// TIA Portal project "SortingLine_Project" (V18)

(* hardware
DEVICE "S7-1200 station_1"  S7-1200 Station
   slot 0: "Rack_0"  S7-1200 Rack  Rack  V1.0
   slot 1: "PLC_Sorting"  CPU 1214C DC/DC/DC  6ES7 214-1AG40-0XB0  V4.6
*)

// ===== PLC "PLC_Sorting"  CPU 1214C DC/DC/DC =====

VAR_GLOBAL   // PLC tag table "Default tag table"
   "start_button" AT %I100.0 : Bool;   // Start push button, NO
   "stop_button" AT %I100.1 : Bool;   // Stop push button, NC
   "emergency_stop" AT %I100.2 : Bool;   // Emergency stop, NC
   "mode_auto" AT %I100.3 : Bool;   // Mode selector, 1 for auto, 0 for manual
   "sensor_entry" AT %I100.4 : Bool;   // Entry sensor, box presence detection
   "sensor_size_low" AT %I100.5 : Bool;   // Low size sensor, detects small boxes
   "sensor_size_high" AT %I100.6 : Bool;   // High size sensor, detects large boxes
   "sensor_left_entry" AT %I100.7 : Bool;   // Pusher 1 retracted limit switch
   "sensor_evac_lane_1" AT %I101.0 : Bool;   // Lane 1 evacuation sensor
   "sensor_evac_lane_2" AT %I101.1 : Bool;   // Lane 2 evacuation sensor
   "light_green" AT %Q0.0 : Bool;   // Green light, machine running
   "light_red" AT %Q0.1 : Bool;   // Red light, machine stopped or fault
   "motor_main_conveyor" AT %Q0.2 : Bool;   // Main conveyor motor
   "motor_lane_1" AT %Q0.3 : Bool;   // Lane 1 conveyor motor
   "motor_lane_2" AT %Q0.4 : Bool;   // Lane 2 conveyor motor
   "pusher_1_command" AT %Q0.5 : Bool;   // Pusher 1 command
   "pusher_2_command" AT %Q0.6 : Bool;   // Pusher 2 command
   "system_running" AT %M0.0 : Bool;   // System running state
   "system_fault" AT %M0.1 : Bool;   // System in fault state
   "box_detected" AT %M0.2 : Bool;   // A box is currently detected
   "box_is_small" AT %M0.3 : Bool;   // Current box is small
   "box_is_large" AT %M0.4 : Bool;   // Current box is large
   "start_pulse" AT %M1.0 : Bool;   // One scan pulse on rising edge of Start_Button
   "edge_start" AT %M1.1 : Bool;   // Edge memory bit for the P_TRIG instruction
   "edge_entry" AT %M1.2 : Bool;
   "edge_evac_lane_1" AT %M1.3 : Bool;
   "edge_evac_lane_2" AT %M1.4 : Bool;
   "entry_pulse" AT %M1.5 : Bool;
   "evac_lane_1_pulse" AT %M1.6 : Bool;
   "evac_lane_2_pulse" AT %M1.7 : Bool;
   "alignment_done" AT %M2.0 : Bool;
   "counter_lane_1" AT %MW10 : Int;
   "counter_lane_2" AT %MW12 : Int;
   "reset_button" AT %I101.2 : Bool;
   "sensor_load_position" AT %I101.3 : Bool;
   "sensor_unload_position" AT %I101.4 : Bool;
   "reset_light" AT %Q0.7 : Bool;
   "motor_feeder" AT %Q1.0 : Bool;
   "light_yellow" AT %Q1.1 : Bool;
   "turn_command" AT %Q1.2 : Bool;
END_VAR

DATA_BLOCK "FB_Mode_Manager_DB"   // DB1
{ S7_Optimized_Access := 'TRUE' }
VERSION : 0.1
// stored: InstanceOfName FB_Mode_Manager
"FB_Mode_Manager"
BEGIN
END_DATA_BLOCK

DATA_BLOCK "FB_Sorting_Logic_DB"   // DB2
{ S7_Optimized_Access := 'TRUE' }
VERSION : 0.1
// stored: InstanceOfName FB_Sorting_Logic
"FB_Sorting_Logic"
BEGIN
END_DATA_BLOCK

DATA_BLOCK "DB_Global"   // DB3
{ S7_Optimized_Access := 'TRUE' }
VERSION : 0.1
BEGIN
END_DATA_BLOCK

// folder: System blocks/Program resources

DATA_BLOCK "Timer_Alignment"   // DB4
{ S7_Optimized_Access := 'TRUE' }
AUTHOR : Simatic
FAMILY : IEC
NAME : IEC_TMR
VERSION : 1.0
// stored: InstanceOfName IEC_TIMER
"IEC_TIMER"
BEGIN
END_DATA_BLOCK

// folder: (top level)

FUNCTION_BLOCK "FB_Mode_Manager"   // FB1, LAD
{ S7_Optimized_Access := 'TRUE' }
VERSION : 0.1
// FB_Mode_Manager
// Purpose: manage safety, mode selection, start and stop logic, indicator lights, main conveyor motor command.
// Inputs: Start_Button, Stop_Button, Emergency_Stop, Mode_Auto
// Outputs: System_Running, System_Fault, Motor_Main_Conveyor, Light_Green, Light_Red
// Author: HoraEmbedded
// Date: 29/09/26
   VAR_TEMP   // added for the SCL form of the ladder/FBD networks
      _w1 : Bool;
   END_VAR
BEGIN

REGION Network 1: Rising edge detection on Start
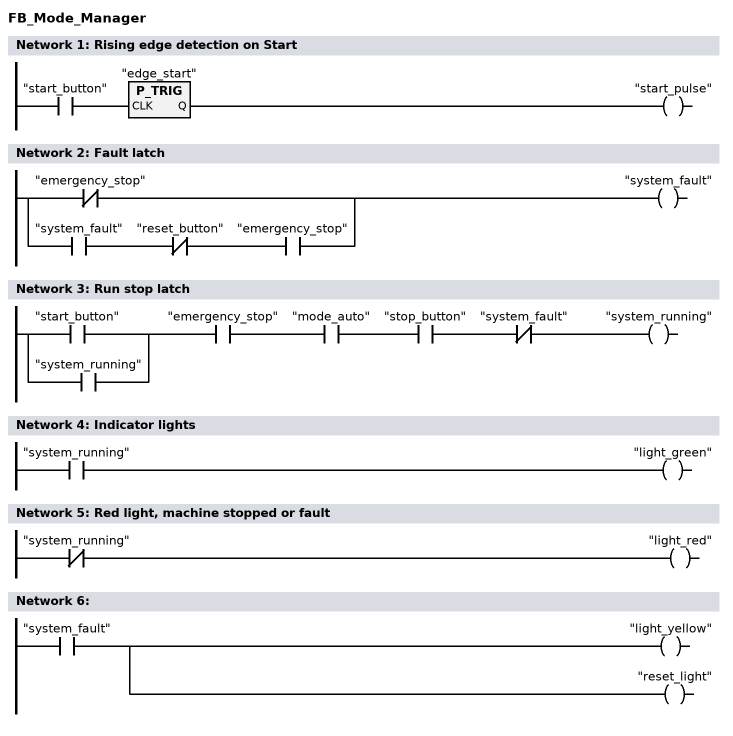
   RUNG wire#powerrail
      Contact( "start_button" )
      P_Trig( "edge_start" )
      Coil( "start_pulse" )
   END_RUNG
   // the same network as SCL:
   #_w1 := "start_button" AND NOT "edge_start";   // rising edge
   "edge_start" := "start_button";
   "start_pulse" := #_w1;
END_REGION

REGION Network 2: Fault latch
   RUNG wire#powerrail
      I_Contact( "emergency_stop" )
      wire#w1
      Coil( "system_fault" )
   END_RUNG
   RUNG wire#powerrail
      Contact( "system_fault" )
      I_Contact( "reset_button" )
      Contact( "emergency_stop" )
   END_RUNG wire#w1
   // the same network as SCL:
   "system_fault" := NOT "emergency_stop" OR ("system_fault" AND NOT "reset_button" AND "emergency_stop");
END_REGION

REGION Network 3: Run stop latch
   RUNG wire#powerrail
      Contact( "start_button" )
      wire#w1
      Contact( "emergency_stop" )
      Contact( "mode_auto" )
      Contact( "stop_button" )
      I_Contact( "system_fault" )
      Coil( "system_running" )
   END_RUNG
   RUNG wire#powerrail
      Contact( "system_running" )
   END_RUNG wire#w1
   // the same network as SCL:
   "system_running" := ("start_button" OR "system_running") AND "emergency_stop" AND "mode_auto" AND "stop_button" AND NOT "system_fault";
END_REGION

REGION Network 4: Indicator lights
   RUNG wire#powerrail
      Contact( "system_running" )
      Coil( "light_green" )
   END_RUNG
   // the same network as SCL:
   "light_green" := "system_running";
END_REGION

REGION Network 5: Red light, machine stopped or fault
   RUNG wire#powerrail
      I_Contact( "system_running" )
      Coil( "light_red" )
   END_RUNG
   // the same network as SCL:
   "light_red" := NOT "system_running";
END_REGION

REGION Network 6
   RUNG wire#powerrail
      Contact( "system_fault" )
      wire#w1
      Coil( "light_yellow" )
   END_RUNG
   RUNG wire#w1
      Coil( "reset_light" )
   END_RUNG
   // the same network as SCL:
   "light_yellow" := "system_fault";
   "reset_light" := "system_fault";
END_REGION
END_FUNCTION_BLOCK

FUNCTION_BLOCK "FB_Sorting_Logic"   // FB2, LAD
{ S7_Optimized_Access := 'TRUE' }
VERSION : 0.1
// FB_Sorting_Logic
// Purpose: detect incoming boxes, classify their size, activate the correct pusher, count evacuated boxes per lane.
// Inputs: Sensor_Entry, Sensor_Size_Low, Sensor_Size_High, Sensor_Evac_Lane_1, Sensor_Evac_Lane_2, System_Running
// Outputs: Pusher_1_Command, Pusher_2_Command
// Internal: Box_Is_Small, Box_Is_Large, Alignment_Done, counters
// Author:HoraEmbedded
// Date: 30/09/2026
   VAR_TEMP   // added for the SCL form of the ladder/FBD networks
      _w1 : Bool;
   END_VAR
BEGIN

REGION Network 1: Rising edge on entry sensor
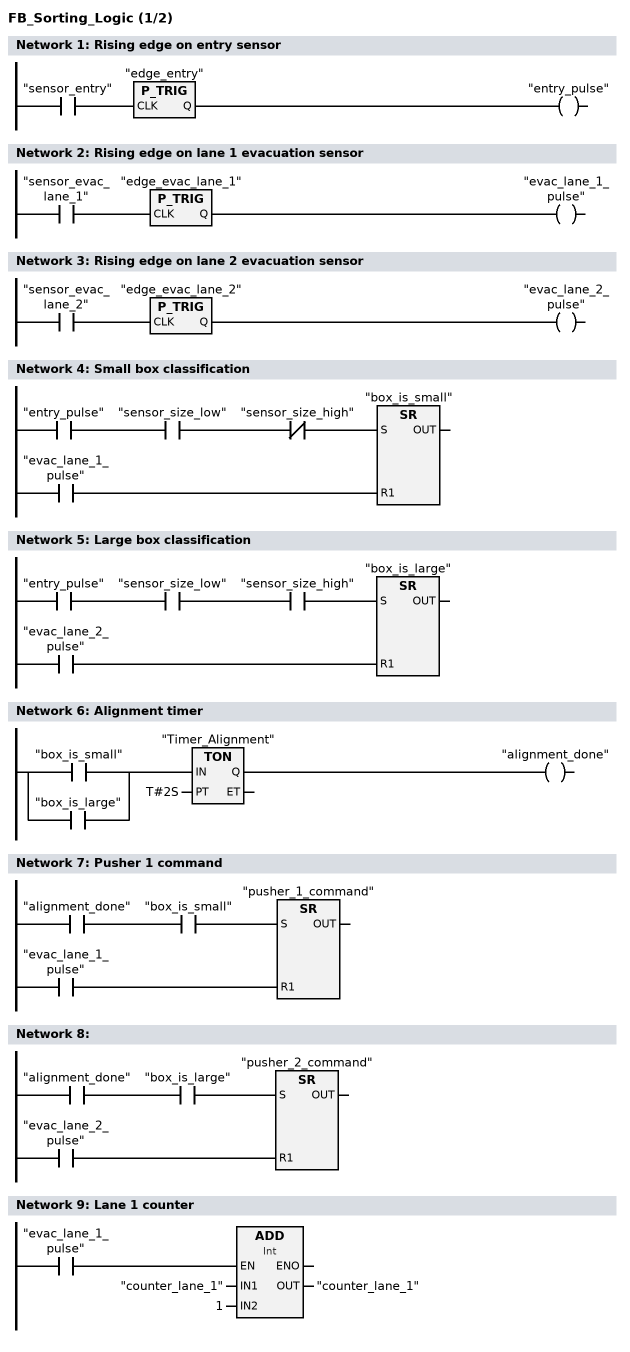
   RUNG wire#powerrail
      Contact( "sensor_entry" )
      P_Trig( "edge_entry" )
      Coil( "entry_pulse" )
   END_RUNG
   // the same network as SCL:
   #_w1 := "sensor_entry" AND NOT "edge_entry";   // rising edge
   "edge_entry" := "sensor_entry";
   "entry_pulse" := #_w1;
END_REGION

REGION Network 2: Rising edge on lane 1 evacuation sensor
   RUNG wire#powerrail
      Contact( "sensor_evac_lane_1" )
      P_Trig( "edge_evac_lane_1" )
      Coil( "evac_lane_1_pulse" )
   END_RUNG
   // the same network as SCL:
   #_w1 := "sensor_evac_lane_1" AND NOT "edge_evac_lane_1";   // rising edge
   "edge_evac_lane_1" := "sensor_evac_lane_1";
   "evac_lane_1_pulse" := #_w1;
END_REGION

REGION Network 3: Rising edge on lane 2 evacuation sensor
   RUNG wire#powerrail
      Contact( "sensor_evac_lane_2" )
      P_Trig( "edge_evac_lane_2" )
      Coil( "evac_lane_2_pulse" )
   END_RUNG
   // the same network as SCL:
   #_w1 := "sensor_evac_lane_2" AND NOT "edge_evac_lane_2";   // rising edge
   "edge_evac_lane_2" := "sensor_evac_lane_2";
   "evac_lane_2_pulse" := #_w1;
END_REGION

REGION Network 4: Small box classification
   RUNG wire#powerrail
      Contact( "entry_pulse" )
      Contact( "sensor_size_low" )
      I_Contact( "sensor_size_high" )
      S_SR(operand := "box_is_small", r1 := wire#w1)
   END_RUNG
   RUNG wire#powerrail
      Contact( "evac_lane_1_pulse" )
   END_RUNG wire#w1
   // the same network as SCL:
   IF "entry_pulse" AND "sensor_size_low" AND NOT "sensor_size_high" THEN
       "box_is_small" := TRUE;   // SR flip-flop
   END_IF;
   IF "evac_lane_1_pulse" THEN "box_is_small" := FALSE; END_IF;
END_REGION

REGION Network 5: Large box classification
   RUNG wire#powerrail
      Contact( "entry_pulse" )
      Contact( "sensor_size_low" )
      Contact( "sensor_size_high" )
      S_SR(operand := "box_is_large", r1 := wire#w1)
   END_RUNG
   RUNG wire#powerrail
      Contact( "evac_lane_2_pulse" )
   END_RUNG wire#w1
   // the same network as SCL:
   IF "entry_pulse" AND "sensor_size_low" AND "sensor_size_high" THEN
       "box_is_large" := TRUE;   // SR flip-flop
   END_IF;
   IF "evac_lane_2_pulse" THEN "box_is_large" := FALSE; END_IF;
END_REGION

REGION Network 6: Alignment timer
   "Timer_Alignment".TON(IN := "box_is_small" OR "box_is_large", PT := T#2S);
   "alignment_done" := "Timer_Alignment".Q;
END_REGION

REGION Network 7: Pusher 1 command
   RUNG wire#powerrail
      Contact( "alignment_done" )
      Contact( "box_is_small" )
      S_SR(operand := "pusher_1_command", r1 := wire#w1)
   END_RUNG
   RUNG wire#powerrail
      Contact( "evac_lane_1_pulse" )
   END_RUNG wire#w1
   // the same network as SCL:
   IF "alignment_done" AND "box_is_small" THEN
       "pusher_1_command" := TRUE;   // SR flip-flop
   END_IF;
   IF "evac_lane_1_pulse" THEN "pusher_1_command" := FALSE; END_IF;
END_REGION

REGION Network 8
   RUNG wire#powerrail
      Contact( "alignment_done" )
      Contact( "box_is_large" )
      S_SR(operand := "pusher_2_command", r1 := wire#w1)
   END_RUNG
   RUNG wire#powerrail
      Contact( "evac_lane_2_pulse" )
   END_RUNG wire#w1
   // the same network as SCL:
   IF "alignment_done" AND "box_is_large" THEN
       "pusher_2_command" := TRUE;   // SR flip-flop
   END_IF;
   IF "evac_lane_2_pulse" THEN "pusher_2_command" := FALSE; END_IF;
END_REGION

REGION Network 9: Lane 1 counter
   RUNG wire#powerrail
      Contact( "evac_lane_1_pulse" )
      { S7_Templates := "SrcType := Int" } Add(in1 := "counter_lane_1", in2 := 1, out => "counter_lane_1")
   END_RUNG
   // the same network as SCL:
   IF "evac_lane_1_pulse" THEN "counter_lane_1" := "counter_lane_1" + 1; END_IF;
END_REGION

REGION Network 10
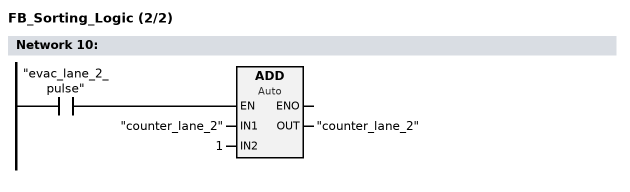
   RUNG wire#powerrail
      Contact( "evac_lane_2_pulse" )
      Add(in1 := "counter_lane_2", in2 := 1, out => "counter_lane_2")
   END_RUNG
   // the same network as SCL:
   IF "evac_lane_2_pulse" THEN "counter_lane_2" := "counter_lane_2" + 1; END_IF;
END_REGION
END_FUNCTION_BLOCK

FUNCTION "FC_IO_Mapping" : Void   // FC1, LAD
{ S7_Optimized_Access := 'TRUE' }
VERSION : 0.1
BEGIN

REGION Network 1: Main conveyor motor
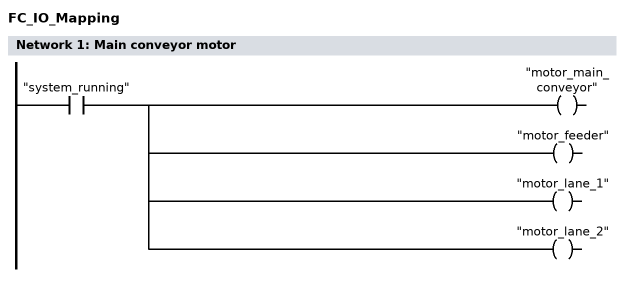
   RUNG wire#powerrail
      Contact( "system_running" )
      wire#w1
      Coil( "motor_main_conveyor" )
   END_RUNG
   RUNG wire#w1
      Coil( "motor_feeder" )
   END_RUNG
   RUNG wire#w1
      Coil( "motor_lane_1" )
   END_RUNG
   RUNG wire#w1
      Coil( "motor_lane_2" )
   END_RUNG
   // the same network as SCL:
   "motor_main_conveyor" := "system_running";
   "motor_feeder" := "system_running";
   "motor_lane_1" := "system_running";
   "motor_lane_2" := "system_running";
END_REGION
END_FUNCTION

FUNCTION "MHJ-PLC-Lab-Function-S71200" : Void   // FC9000, SCL
{ S7_Optimized_Access := 'TRUE' }
VERSION : 0.1
   VAR_TEMP
      rdTimeReturn : Int;
      outputTime : DTL;
      SyncVal : Byte;
      forVal : Int;
      forVal_2 : Int;
      Value : Byte;
   END_VAR
   VAR CONSTANT
      CompVal : Byte := 16#34;
      Value_01 : Byte := 16#11;
      Value_01_DW : DWord := 16#A165_D992;
      Value_02_DW : DWord := 16#58BE_4401;
   END_VAR
BEGIN

   #Value:=PEEK(area := 16#82,
        dbNumber := 0,
        byteOffset := 511);
   #Value := #Value + 1;

   POKE(area := 16#82,
        dbNumber := 0,
        byteOffset := 511,
        value := #Value);

   POKE(area:=16#81,
        dbNumber:=0,
        byteOffset:=1016,
        value:=#Value_01_DW);
   POKE(area := 16#81,
        dbNumber := 0,
        byteOffset := 1020,
        value := #Value_02_DW);

   POKE(area := 16#81,
        dbNumber := 0,
        byteOffset := 511,
        value := B#16#00);

   FOR #forVal := 0 TO 120 DO
       FOR #forVal_2:=0 TO 10 DO
           #rdTimeReturn:=RD_SYS_T(#outputTime);
           #rdTimeReturn := WR_SYS_T(#outputTime);
           #rdTimeReturn := RD_SYS_T(#outputTime);
           #rdTimeReturn := WR_SYS_T(#outputTime);
       END_FOR;
       #SyncVal:= PEEK(area := 16#81,
                      dbNumber := 0,
                      byteOffset := 511);
       IF #SyncVal = #CompVal THEN
          GOTO M_1;
       END_IF;
   END_FOR;
   RETURN;

   M_1:
   POKE(area := 16#81,
        dbNumber := 0,
        byteOffset := 511,
        value := B#16#0);
END_FUNCTION

ORGANIZATION_BLOCK "Main"   // OB1, LAD, ProgramCycle
TITLE = "Main Program Sweep (Cycle)"
{ S7_Optimized_Access := 'TRUE' }
VERSION : 0.1
   VAR_INPUT
      Initial_Call : Bool;   // Initial call of this OB
      Remanence : Bool;   // =True, if remanent data are available
   END_VAR
BEGIN

REGION Network 1
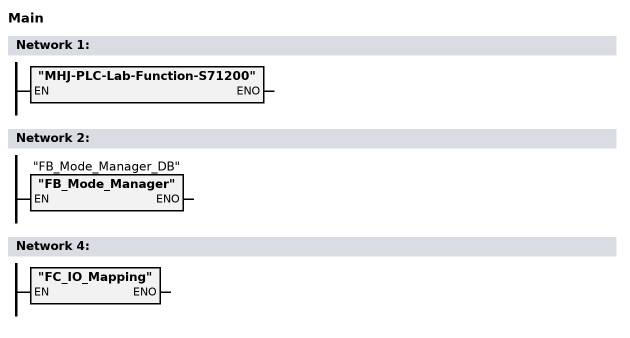
   RUNG wire#powerrail
      "MHJ-PLC-Lab-Function-S71200"()
   END_RUNG
   // the same network as SCL:
   "MHJ-PLC-Lab-Function-S71200"();
END_REGION

REGION Network 2
   RUNG wire#powerrail
      "FB_Mode_Manager_DB"()
   END_RUNG
   // the same network as SCL:
   "FB_Mode_Manager_DB"();   // "FB_Mode_Manager"
END_REGION

REGION Network 4
   RUNG wire#powerrail
      "FC_IO_Mapping"()
   END_RUNG
   // the same network as SCL:
   "FC_IO_Mapping"();
END_REGION
END_ORGANIZATION_BLOCK